PROGRAM TelescopeAuxiliary
VAR
	MQTTTimer : TON := (PT:=T#5S);
	pressure_voltage:	REAL;
END_VAR
VAR_OUTPUT
	// BT9 mirror
	temperature_mirror2:	REAL;
	// BT10
	temperature_mirror1:	REAL;
	// BT11
	temperature_mirror3:	REAL;
	// BT12
	temperature_tube:		REAL;
	// BT13
	temperature_bearing1:	REAL;
	// BT14
	temperature_bearing2:	REAL;

	// dewar pressure 0..10V Pfeiffer 
	pressure_Dewar:	REAL;
	// dewar temperature PT100
	temperature_Dewar:	REAL;
	

END_VAR

temperature_mirror2 := GVL_Telescope.temperature_mirror2 / 100.0;
temperature_mirror1 := GVL_Telescope.temperature_mirror1 / 100.0;
temperature_mirror3 := GVL_Telescope.temperature_mirror3 / 100.0;
temperature_tube 	:= GVL_Telescope.temperature_tube / 100.0;
temperature_bearing1 := GVL_Telescope.temperature_bearing1 / 100.0;
temperature_bearing2 := GVL_Telescope.temperature_bearing2 / 100.0;

MQTTTimer(IN:=TRUE);
IF MQTTTimer.Q THEN // publish new payload every second

	MAIN.MQTTClient.Publish('telescope', 'dome',  'Mirror2Temperature',	LREAL_TO_FMTSTR(temperature_mirror2, 2, TRUE));
	MAIN.MQTTClient.Publish('telescope', 'dome', 'Mirror1Temperature',	LREAL_TO_FMTSTR(temperature_mirror1, 2, TRUE));
	IF GVL_Telescope.temperature_mirror3>0 AND GVL_Telescope.temperature_mirror3<32767 THEN
		MAIN.MQTTClient.Publish('telescope', 'dome', 'Mirror3Temperature',	LREAL_TO_FMTSTR(temperature_mirror3, 2, TRUE));
	END_IF
	IF GVL_Telescope.temperature_tube>0 AND GVL_Telescope.temperature_tube<32767 THEN
		MAIN.MQTTClient.Publish('telescope', 'dome', 'TubeTemperature', 	LREAL_TO_FMTSTR(temperature_tube, 2, TRUE));
	END_IF
	IF GVL_Telescope.temperature_bearing1>0 AND GVL_Telescope.temperature_bearing1<32767 THEN
		MAIN.MQTTClient.Publish('telescope', 'dome', 'Bearing1Temperature', LREAL_TO_FMTSTR(temperature_bearing1, 2, TRUE));
	END_IF
	IF GVL_Telescope.temperature_bearing2>0 AND GVL_Telescope.temperature_bearing2<32767 THEN
		MAIN.MQTTClient.Publish('telescope', 'dome', 'Bearing2Temperature', LREAL_TO_FMTSTR(temperature_bearing2, 2, TRUE));
	END_IF
	
	MAIN.MQTTClient.Publish('telescope', 'instrument', 'DewarPressureVoltage',	LREAL_TO_FMTSTR(pressure_voltage, 3, TRUE));
	IF NOT GVL_Auxiliary.Dewar_temperature_error THEN
		MAIN.MQTTClient.Publish('telescope', 'instrument', 'DewarTemperature',	LREAL_TO_FMTSTR(temperature_Dewar, 2, TRUE));
	END_IF
	IF pressure_voltage > 0.001 THEN
		MAIN.MQTTClient.Publish('telescope', 'instrument', 'DewarPressure',	LREAL_TO_FMTSTR(pressure_Dewar, 2, TRUE));
	END_IF
	
	MQTTTimer(IN:=FALSE);

END_IF

END_PROGRAM

(* stored: Version 1.1.0.1, ProductVersion 3.1.4024.9
   POU TelescopeAuxiliary: Id {974ce34a-6026-4bc5-b92d-99da70a09948}, SpecialFunc None *)
